FUNCTION_BLOCK FB_PlanarMover

VAR_INPUT
	nMoverId			: UDINT;
	iTcIoXtsXpuMover	: I_TcIoXtsXpuMover;
END_VAR

VAR
	_McPlanarMover	: MC_PlanarMover;
	_PlanarTrail    : MC_PlanarTrackTrail;
  	

END_VAR

PROPERTY IsCommandedInShortcut : BOOL
GET
VAR
	nCounter: UDINT := 0;
END_VAR
_mcPlanarMover.GetTrackTrailInformation(_PlanarTrail);

IF  _PlanarTrail.Size > 1 THEN
	FOR nCounter := 1 TO _PlanarTrail.Size  DO
		IF _PlanarTrail.GetTrackOidAt(nCounter) = GVL_Mc3.MC_Tracks[E_Tracknum.Small].MCTOPLC_STD.TrackOID  THEN
			IsCommandedInShortcut := TRUE;
		END_IF
	END_FOR
END_IF
END_GET
SET
END_SET
END_PROPERTY

METHOD JoinTrack

VAR_INPUT
	feedback: REFERENCE TO MC_PlanarFeedback;
END_VAR

VAR_IN_OUT
	track: MC_PlanarTrack;
END_VAR
_McPlanarMover.JoinTrack(feedback, track, 0, 0);
END_METHOD

PROPERTY McPlanarMover : REFERENCE TO MC_PlanarMover
GET
McPlanarMover ref= _McPlanarMover;
END_GET
END_PROPERTY

METHOD Update : PVOID
_mcPlanarMover.Update();


_mcPlanarMover.GetTrackTrailInformation(_PlanarTrail);

IF(* _PlanarTrail.Error OR*) _PlanarTrail.Size < 1 THEN
   RETURN;
END_IF
   
//SmallCircle
IF _PlanarTrail.GetTrackOidAt(2) = MC_Tracks[E_TrackNum.Small].MCTOPLC_STD.TrackOID   THEN
	iTcIoXtsXpuMover.SetActiveTrackObjectId(XtsShortcutOid);
//BigCircle
ELSIF _PlanarTrail.GetTrackOidAt(2) =MC_Tracks[E_TrackNum.Big].MCTOPLC_STD.TrackOID THEN
	iTcIoXtsXpuMover.SetActiveTrackObjectId(XtsOutterLoopOid);
END_IF
END_METHOD

END_FUNCTION_BLOCK

(* stored: Version 1.1.0.1, ProductVersion 3.1.4024.12
   POU FB_PlanarMover: Id {e98e5f10-cdde-43fc-96da-1ae5f511366a}, SpecialFunc None
   Folder Methods: Id {497e6300-3e6d-49b8-a318-13b94b960f56}
   Folder Properties: Id {bafe569f-b5f0-4de9-ae48-854cd11ccd2e}
   Property IsCommandedInShortcut: Id {e5e69e7e-f163-4728-82da-b10e582ce622}
   Get Get: Id {7a71ba46-249d-415a-b1f4-f1c52c07bed0}
   Set Set: Id {53913d7d-2725-41d6-8d63-9e6898f391bc}
   Method JoinTrack: Id {fd819ce6-c064-4bae-aa84-926325f13c12}
   Property McPlanarMover: Id {79d72b75-52b9-47c8-886e-5e60276bf5f1}
   Get Get: Id {71cad725-c4c4-49c5-9410-cee17b681f5a}
   Method Update: Id {2a189ea7-97f2-4dc0-980a-fdde9c091766} *)
